# EPICS substitutions: apps/jscalerApp/Db/jscalers_TDCFTOF4_TRIG.substitutions
file "db/jscaler_channel_DISC.db" {
pattern { CrNo,CrName,Sl,Ch,Det,Sys,Element,CScode,ThreshTRG,ThreshTDC,Mode,Counts }
{ "05","TDCFTOF4","20","15","TRIG","DISC","SEC4_F00","0x1405","0xF","0x10F","0x10F","0xF" }
}
